INTERFACE ITF_BaseTopElement_HMI_Connector_View EXTENDS ITF_BaseGroupElement_HMI_Connector_View

END_INTERFACE

(* stored: Version 1.1.0.1
   Itf ITF_BaseTopElement_HMI_Connector_View: Id {770e6841-0e75-097b-268d-045557e39b52} *)
